Omron CX-Programmer project NewProject (CX-Programmer 9.63)

# PLC Projet_Chaine_Auto: CP1L-E EM

## Global symbols (name address type ; comment)
0.00 BOOL  ; I: Emergency Stop
100.04 BOOL  ; O:ON/OFF
D2 CHANNEL  ; password
D4 CHANNEL  ; Software version
D5 CHANNEL  ; Control the indirect window to display
D6 CHANNEL  ; Control screen N° to display
H30.08 BOOL  ; 0search: 0 search completed
H5 CHANNEL  ; Screen word
H99.00 BOOL  ; E STOP
W0.00 BOOL  ; WO: reload save value of PV pulse output
W111.00 BOOL  ; Interlock axis 0
W15.00 BOOL  ; PB: On/OFF
W15.01 BOOL  ; PB: ON OFF
W500.00 BOOL  ; MF ON

## Program NewProgram1 (cyclic task 0)

### Section ON_OFF

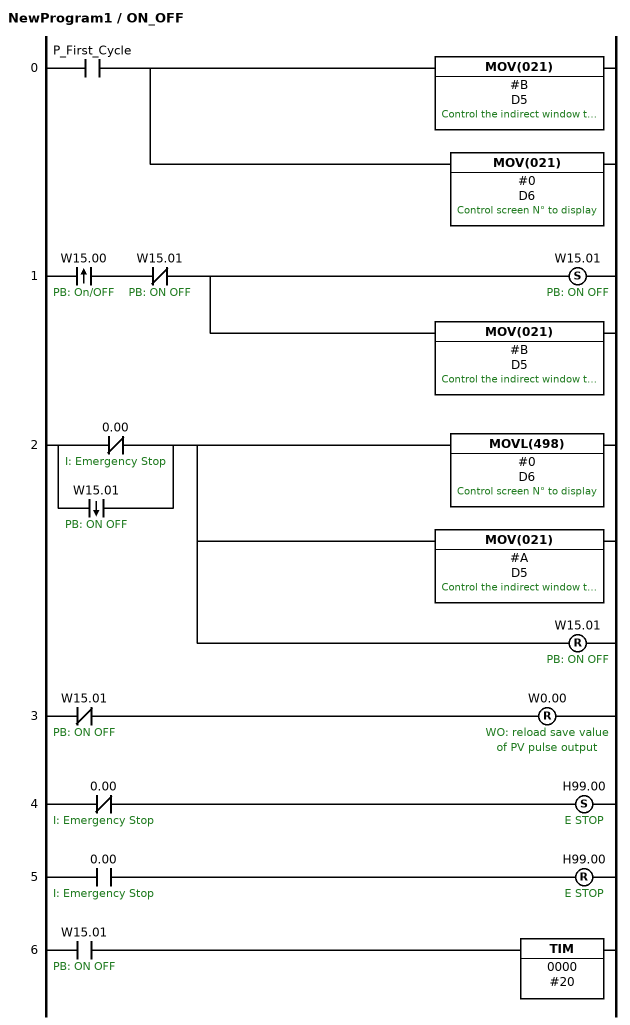
; rung 0
LD P_First_Cycle
MOV(021) #B D5  ; Control the indirect window to display
MOV(021) #0 D6  ; Control screen N° to display
; rung 1
@LD W15.00  ; PB: On/OFF
ANDNOT W15.01  ; PB: ON OFF
SET W15.01  ; PB: ON OFF
MOV(021) #B D5  ; Control the indirect window to display
; rung 2
LDNOT 0.00  ; I: Emergency Stop
%OR W15.01  ; PB: ON OFF
MOVL(498) #0 D6  ; Control screen N° to display
MOV(021) #A D5  ; Control the indirect window to display
RSET W15.01  ; PB: ON OFF
; rung 3
LDNOT W15.01  ; PB: ON OFF
RSET W0.00  ; WO: reload save value of PV pulse output
; rung 4
LDNOT 0.00  ; I: Emergency Stop
SET H99.00  ; E STOP
; rung 5
LD 0.00  ; I: Emergency Stop
RSET H99.00  ; E STOP
; rung 6
LD W15.01  ; PB: ON OFF
TIM 0000 #20

### Section STOP

### Section SCREEN

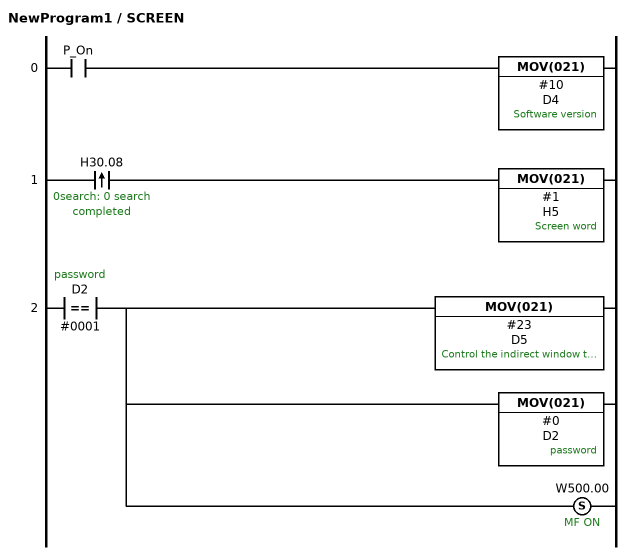
; rung 0
LD P_On
MOV(021) #10 D4  ; Software version
; rung 1
@LD H30.08  ; 0search: 0 search completed
MOV(021) #1 H5  ; Screen word
; rung 2
LD=(300) D2 #0001  ; password
MOV(021) #23 D5  ; Control the indirect window to display
MOV(021) #0 D2  ; password
SET W500.00  ; MF ON

### Section CYCLE

### Section AXIS_1
; rung 0: Axe pour la partie xxxxx de la chaine

### Section AXIS_2
; rung 0: Axe pour la partie xxxxx de la chaine

### Section AXIS_3
; rung 0: Axe pour la partie xxxxx de la chaine

### Section ANIMATION_SCREEN_1
; rung 0: Animation pour la page de xxxxxx de la chaine

### Section ANIMATION_SCREEN_2
; rung 0: Animation pour la page de xxxxxx de la chaine

### Section ANIMATION_SCREEN_3
; rung 0: Animation pour la page de xxxxxx de la chaine

### Section Output

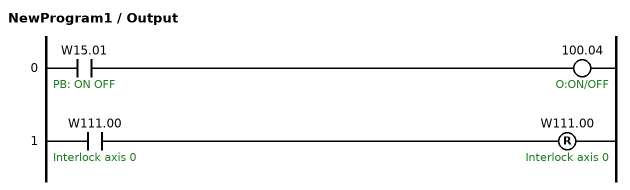
; rung 0
LD W15.01  ; PB: ON OFF
OUT 100.04  ; O:ON/OFF
; rung 1
LD W111.00  ; Interlock axis 0
RSET W111.00  ; Interlock axis 0

### Section END
; rung 0
END(001)